Fanuc KAREL source: kb00078.KL

-- PROVISIONAL review KL for V770-1; original PC SHA256 f9a7c42a7141df73bd189d7dea33463bceb4e77cf34643e8ba57b3f210e6ae5b
-- Incomplete behavior may be omitted. Consult companion uncertainty JSON. Do not deploy.
PROGRAM KB00078
%NOLOCKGROUP
BEGIN
  -- UNRESOLVED_PC offsets 5-21; opcodes 27,22,31,23
  -- UNRESOLVED_PC offsets 26-30; opcodes 7F
END KB00078
